TYPE DSV2_A1_ArmPnpSequenceCall : (*Full Occupied Byte = 1700*)
STRUCT

	bEnableCallArmNo 					: BOOL; (* Byte "n" *)
	bCallSt								: BOOL; (* Byte "n+1" *)

	bCallCompleted 						: BOOL; (* Byte "n+2" *)
	bInvalidProductRecipeNoErrHold		: BOOL; (* Byte "n+3" *)
	bInvalidProductRecipeNoErrPulse	: BOOL; (* Byte "n+4" *)
	bInvalidProductRecipeStepErrHold 	: BOOL; (* Byte "n+5" *)
	bInvalidProductRecipeStepErrPulse	: BOOL; (* Byte "n+6" *)
	bCallUpDownPatternMemoryErr 		: BOOL; (* Byte "n+7" *)
	bCallArmSpeedProfileMemoryErr 	: BOOL; (* Byte "n+8" *)
	bCallPickStationNoErr 				: BOOL; (* Byte "n+9" *)
	bCallTransferStationNoErr 			: BOOL; (* Byte "n+10" *)

	sReservedBool 						: STRING(88); (* Byte "n+11~n+99" *)

	iCallArmNo 							: INT; (* Byte "n+100~n+101" *)
	iProductRecipeNoCall 				: INT; (* Byte "n+102~n+103" *)
	iProductRecipeStepCall				: INT; (* Byte "n+104~n+105" *)
	iCalledProductRecipeNo 				: INT; (* Byte "n+106~n+107" *) (*New*)
	iCalledProductRecipeStep			: INT; (* Byte "n+108~n+109" *) (*New*)

	sReservedInt 							: STRING(89); (* Byte "n+110~n+199" *)

	sProductRecipeDescription 			: STRING(50);


	DSGnrCalledArmPnpParameter 		: DSV2_Gnr_CalledArmPnpParameter;



END_STRUCT
END_TYPE

(* stored: Version 1.1.0.1, ProductVersion 3.1.4024.12
   DUT DSV2_A1_ArmPnpSequenceCall: Id {8fa5adaf-c51f-4a8e-90af-a4ece95c5fb1} *)
